// TIA Portal V16 export
// export: Created 2025-05-30T16:35:50.2365001Z, ExportSetting WithDefaults, DisplayName Totally Integrated Automation Portal, DisplayVersion V16, DisplayName TIA Portal Version Control Interface, DisplayVersion V16, DisplayName TIA Portal Openness, DisplayVersion V16, DisplayName STEP 7 Professional, DisplayVersion V16, DisplayName STEP 7 Safety, DisplayVersion V16, DisplayName WinCC Advanced, DisplayVersion V16
FUNCTION "1 - Outputs" : Void   // FC5, LAD
VERSION : 0.1
// This Function program is for operating the machine automatic and manual.
// stored: AutoNumber true, IsIECCheckEnabled false, UDAEnableTagReadback false
   VAR_TEMP
      Valve_2_Pulse : Bool;
      BlowOff_Activated : Bool;
      BlowOffManual : Bool;
      Pulse1 : Bool;
   END_VAR
   VAR_TEMP   // added for the SCL form of the ladder/FBD networks
      _w1 : Bool;
   END_VAR
BEGIN

REGION Network 1: Drive 1 - Control
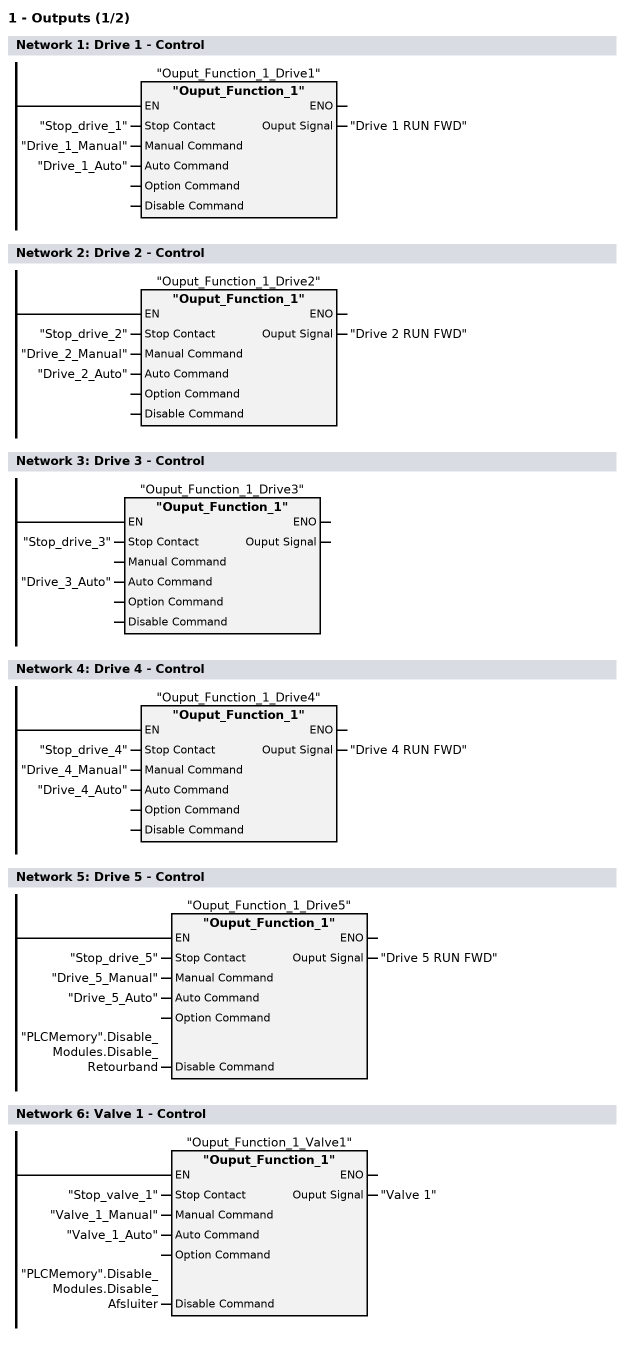
   RUNG wire#powerrail
      "Ouput_Function_1_Drive1"("Stop Contact" := "Stop_drive_1", "Manual Command" := "Drive_1_Manual", "Auto Command" := "Drive_1_Auto", "Option Command" :=, "Disable Command" :=, "Ouput Signal" => "Drive 1 RUN FWD")
   END_RUNG
   // the same network as SCL:
   "Ouput_Function_1_Drive1"("Stop Contact" := "Stop_drive_1",   // "Ouput_Function_1"
                           "Manual Command" := "Drive_1_Manual",
                           "Auto Command" := "Drive_1_Auto",
                           "Ouput Signal" => "Drive 1 RUN FWD");
END_REGION

REGION Network 2: Drive 2 - Control
   RUNG wire#powerrail
      "Ouput_Function_1_Drive2"("Stop Contact" := "Stop_drive_2", "Manual Command" := "Drive_2_Manual", "Auto Command" := "Drive_2_Auto", "Option Command" :=, "Disable Command" :=, "Ouput Signal" => "Drive 2 RUN FWD")
   END_RUNG
   // the same network as SCL:
   "Ouput_Function_1_Drive2"("Stop Contact" := "Stop_drive_2",   // "Ouput_Function_1"
                           "Manual Command" := "Drive_2_Manual",
                           "Auto Command" := "Drive_2_Auto",
                           "Ouput Signal" => "Drive 2 RUN FWD");
END_REGION

REGION Network 3: Drive 3 - Control
   RUNG wire#powerrail
      "Ouput_Function_1_Drive3"("Stop Contact" := "Stop_drive_3", "Manual Command" :=, "Auto Command" := "Drive_3_Auto", "Option Command" :=, "Disable Command" :=, "Ouput Signal" =>)
   END_RUNG
   // the same network as SCL:
   "Ouput_Function_1_Drive3"("Stop Contact" := "Stop_drive_3", "Auto Command" := "Drive_3_Auto");   // "Ouput_Function_1"
END_REGION

REGION Network 4: Drive 4 - Control
   RUNG wire#powerrail
      "Ouput_Function_1_Drive4"("Stop Contact" := "Stop_drive_4", "Manual Command" := "Drive_4_Manual", "Auto Command" := "Drive_4_Auto", "Option Command" :=, "Disable Command" :=, "Ouput Signal" => "Drive 4 RUN FWD")
   END_RUNG
   // the same network as SCL:
   "Ouput_Function_1_Drive4"("Stop Contact" := "Stop_drive_4",   // "Ouput_Function_1"
                           "Manual Command" := "Drive_4_Manual",
                           "Auto Command" := "Drive_4_Auto",
                           "Ouput Signal" => "Drive 4 RUN FWD");
END_REGION

REGION Network 5: Drive 5 - Control
   RUNG wire#powerrail
      "Ouput_Function_1_Drive5"("Stop Contact" := "Stop_drive_5", "Manual Command" := "Drive_5_Manual", "Auto Command" := "Drive_5_Auto", "Option Command" :=, "Disable Command" := "PLCMemory".Disable_Modules.Disable_Retourband, "Ouput Signal" => "Drive 5 RUN FWD")
   END_RUNG
   // the same network as SCL:
   "Ouput_Function_1_Drive5"("Stop Contact" := "Stop_drive_5",   // "Ouput_Function_1"
                           "Manual Command" := "Drive_5_Manual",
                           "Auto Command" := "Drive_5_Auto",
                           "Disable Command" := "PLCMemory".Disable_Modules.Disable_Retourband,
                           "Ouput Signal" => "Drive 5 RUN FWD");
END_REGION

REGION Network 6: Valve 1 - Control
   RUNG wire#powerrail
      "Ouput_Function_1_Valve1"("Stop Contact" := "Stop_valve_1", "Manual Command" := "Valve_1_Manual", "Auto Command" := "Valve_1_Auto", "Option Command" :=, "Disable Command" := "PLCMemory".Disable_Modules.Disable_Afsluiter, "Ouput Signal" => "Valve 1")
   END_RUNG
   // the same network as SCL:
   "Ouput_Function_1_Valve1"("Stop Contact" := "Stop_valve_1",   // "Ouput_Function_1"
                           "Manual Command" := "Valve_1_Manual",
                           "Auto Command" := "Valve_1_Auto",
                           "Disable Command" := "PLCMemory".Disable_Modules.Disable_Afsluiter,
                           "Ouput Signal" => "Valve 1");
END_REGION

REGION Network 7: Valve 2 - Control
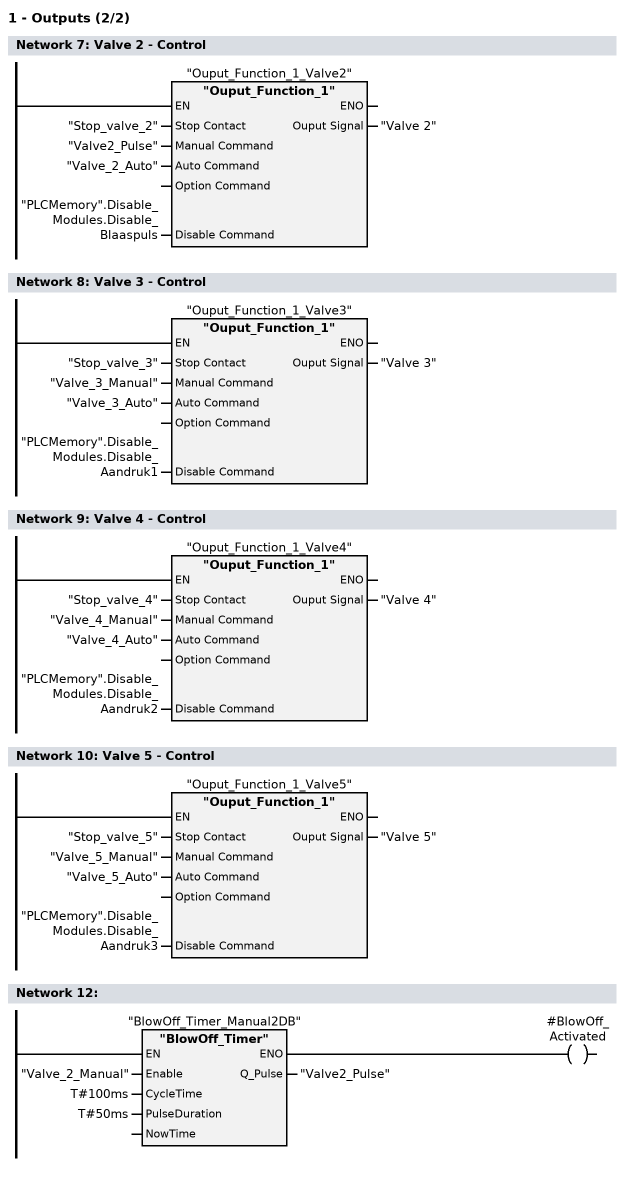
   RUNG wire#powerrail
      "Ouput_Function_1_Valve2"("Stop Contact" := "Stop_valve_2", "Manual Command" := "Valve2_Pulse", "Auto Command" := "Valve_2_Auto", "Option Command" :=, "Disable Command" := "PLCMemory".Disable_Modules.Disable_Blaaspuls, "Ouput Signal" => "Valve 2")
   END_RUNG
   // the same network as SCL:
   "Ouput_Function_1_Valve2"("Stop Contact" := "Stop_valve_2",   // "Ouput_Function_1"
                           "Manual Command" := "Valve2_Pulse",
                           "Auto Command" := "Valve_2_Auto",
                           "Disable Command" := "PLCMemory".Disable_Modules.Disable_Blaaspuls,
                           "Ouput Signal" => "Valve 2");
END_REGION

REGION Network 8: Valve 3 - Control
   RUNG wire#powerrail
      "Ouput_Function_1_Valve3"("Stop Contact" := "Stop_valve_3", "Manual Command" := "Valve_3_Manual", "Auto Command" := "Valve_3_Auto", "Option Command" :=, "Disable Command" := "PLCMemory".Disable_Modules.Disable_Aandruk1, "Ouput Signal" => "Valve 3")
   END_RUNG
   // the same network as SCL:
   "Ouput_Function_1_Valve3"("Stop Contact" := "Stop_valve_3",   // "Ouput_Function_1"
                           "Manual Command" := "Valve_3_Manual",
                           "Auto Command" := "Valve_3_Auto",
                           "Disable Command" := "PLCMemory".Disable_Modules.Disable_Aandruk1,
                           "Ouput Signal" => "Valve 3");
END_REGION

REGION Network 9: Valve 4 - Control
   RUNG wire#powerrail
      "Ouput_Function_1_Valve4"("Stop Contact" := "Stop_valve_4", "Manual Command" := "Valve_4_Manual", "Auto Command" := "Valve_4_Auto", "Option Command" :=, "Disable Command" := "PLCMemory".Disable_Modules.Disable_Aandruk2, "Ouput Signal" => "Valve 4")
   END_RUNG
   // the same network as SCL:
   "Ouput_Function_1_Valve4"("Stop Contact" := "Stop_valve_4",   // "Ouput_Function_1"
                           "Manual Command" := "Valve_4_Manual",
                           "Auto Command" := "Valve_4_Auto",
                           "Disable Command" := "PLCMemory".Disable_Modules.Disable_Aandruk2,
                           "Ouput Signal" => "Valve 4");
END_REGION

REGION Network 10: Valve 5 - Control
   RUNG wire#powerrail
      "Ouput_Function_1_Valve5"("Stop Contact" := "Stop_valve_5", "Manual Command" := "Valve_5_Manual", "Auto Command" := "Valve_5_Auto", "Option Command" :=, "Disable Command" := "PLCMemory".Disable_Modules.Disable_Aandruk3, "Ouput Signal" => "Valve 5")
   END_RUNG
   // the same network as SCL:
   "Ouput_Function_1_Valve5"("Stop Contact" := "Stop_valve_5",   // "Ouput_Function_1"
                           "Manual Command" := "Valve_5_Manual",
                           "Auto Command" := "Valve_5_Auto",
                           "Disable Command" := "PLCMemory".Disable_Modules.Disable_Aandruk3,
                           "Ouput Signal" => "Valve 5");
END_REGION

REGION Network 11: Blow Off Manual
END_REGION

REGION Network 12
   RUNG wire#powerrail
      "BlowOff_Timer_Manual2DB"(Enable := "Valve_2_Manual", CycleTime := T#100ms, PulseDuration := T#50ms, NowTime :=, Q_Pulse => "Valve2_Pulse")
      Coil( #BlowOff_Activated )
   END_RUNG
   // the same network as SCL:
   "BlowOff_Timer_Manual2DB"(Enable := "Valve_2_Manual",   // "BlowOff_Timer"
                           CycleTime := T#100ms,
                           PulseDuration := T#50ms,
                           Q_Pulse => "Valve2_Pulse",
                           ENO => #_w1);
   #BlowOff_Activated := #_w1;
END_REGION
END_FUNCTION
